TYPE (* A Structured Data Type *)
  (* Standard: 61499-2 *)
  (* Version 0.1, 2003-12-05, JHC, Rockwell Automation, Renamed from NEWSTRUCT. *)
  (* Version 0.0, 2000-05-27, JHC, Rockwell Automation *)
  (* Compiler header: package fb.rt.template; *)
  (* ASN.1 tag PRIVATE 5 *)
  Structured : STRUCT
    VAR1 : BOOL;
    VAR2 : INT;
  END_STRUCT;
END_TYPE
